// TIA Portal project "Traffic_light_Control" (V13)

(* hardware
DEVICE "S7300/ET200M station_1"  S7-300 station
   slot 0: "Rail_0"  Rail  6ES7 390-1***0-0AA0
   slot 2: "PLC_1"  CPU 314C-2 PN/DP  6ES7 314-6EH04-0AB0  V3.3
      slot 2: "PROFINET interface_1"  PN-IO
         slot 1: "Port_1"  Port
         slot 2: "Port_2"  Port
      slot 5: "DI 24/DO 16_1"  DI24/DO16
      slot 6: "AI 5/AO 2_1"  AI5/AO2
      slot 7: "Count_1"  Counter
      slot 8: "Positioning_1"  Positioning
*)

// ===== PLC "PLC_1"  CPU 314C-2 PN/DP =====

VAR_GLOBAL   // PLC tag table "Default tag table"
   "Start" AT %I0.0 : Bool;
   "Operation_System" AT %M0.0 : Bool;
   "Stop" AT %I0.1 : Bool;
   "Green_Light" AT %Q0.0 : Bool;
   "Yellow_Light" AT %Q0.1 : Bool;
   "Red_Light" AT %Q0.2 : Bool;
END_VAR

ORGANIZATION_BLOCK "Main"   // OB1, LAD
TITLE = "Main Program Sweep (Cycle)"
{ S7_Optimized_Access := 'FALSE' }
VERSION : 0.1
   VAR_TEMP
      OB1_EV_CLASS : Byte;   // Bits 0-3 = 1 (Coming event), Bits 4-7 = 1 (Event class 1)
      OB1_SCAN_1 : Byte;   // 1 (Cold restart scan 1 of OB 1), 3 (Scan 2-n of OB 1)
      OB1_PRIORITY : Byte;   // Priority of OB Execution
      OB1_OB_NUMBR : Byte;   // 1 (Organization block 1, OB1)
      OB1_RESERVED_1 : Byte;   // Reserved for system
      OB1_RESERVED_2 : Byte;   // Reserved for system
      OB1_PREV_CYCLE : Int;   // Cycle time of previous OB1 scan (milliseconds)
      OB1_MIN_CYCLE : Int;   // Minimum cycle time of OB1 (milliseconds)
      OB1_MAX_CYCLE : Int;   // Maximum cycle time of OB1 (milliseconds)
      OB1_DATE_TIME : Date_And_Time;   // Date and time OB1 started
   END_VAR
BEGIN

REGION Network 1
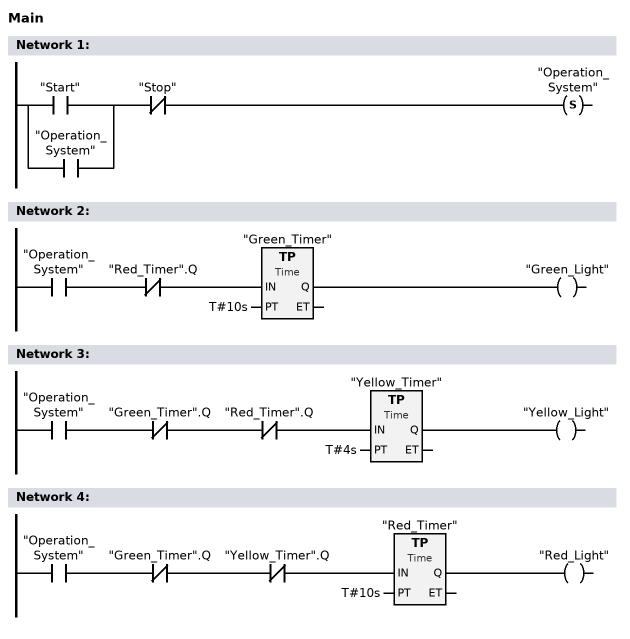
   RUNG wire#powerrail
      Contact( "Start" )
      wire#w1
      I_Contact( "Stop" )
      S_Coil( "Operation_System" )
   END_RUNG
   RUNG wire#powerrail
      Contact( "Operation_System" )
   END_RUNG wire#w1
   // the same network as SCL:
   IF ("Start" OR "Operation_System") AND NOT "Stop" THEN "Operation_System" := TRUE; END_IF;
END_REGION

REGION Network 2
   "Green_Timer".TP(IN := "Operation_System" AND NOT "Red_Timer".Q, PT := T#10s);
   "Green_Light" := "Green_Timer".Q;
END_REGION

REGION Network 3
   "Yellow_Timer".TP(IN := "Operation_System" AND NOT "Green_Timer".Q AND NOT "Red_Timer".Q, PT := T#4s);
   "Yellow_Light" := "Yellow_Timer".Q;
END_REGION

REGION Network 4
   "Red_Timer".TP(IN := "Operation_System" AND NOT "Green_Timer".Q AND NOT "Yellow_Timer".Q, PT := T#10s);
   "Red_Light" := "Red_Timer".Q;
END_REGION
END_ORGANIZATION_BLOCK